// TIA Portal V20 export
TYPE "type_emRelations_em9_cmStatus"
// stored: Access Published, Namespace Unit1
   STRUCT
      VisionJRDetect : "LBC_typeDigitalSignalControlNode";
      VisionStageLiftUpDown : "LBC_typeTwoWayActuatorControlNode";
      VisionLightUpDown : "LBC_typeTwoWayActuatorControlNode";
      VisionControl : "LER_typeVisionControlNode";
   END_STRUCT;
END_TYPE
